TEXTLIST Alarm_TextList
  1 = 'Power Interrupted Fault'
  2 = 'Test 1'
  3 = 'Test 2'
  4 = 'Test 3'
  5 = 'Test 4'
   = ''
END_TEXTLIST

(* stored: Version 1.1.0.1
   TextList Alarm_TextList: Id {9f1faf1c-efde-4b0a-9f66-57a2cf575857} *)
